ABB RobotStudio station: IndustrialFinal_1.3.rspag

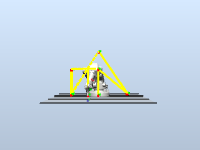
--- station ---
Station IndustrialFinal_1 (saved by RobotStudio 6.5.7558.2005)
Controller IRB_1600_8kg_1.2m
  mechanical unit ROB_1: IRB1600_8_120__02, 6 joints, base frame (0, 0, 0) mm
Layout (positions relative to the parent item):
  - IRB1600_8_120__02 [mechanism, from Robots\IRB1600_8_120_G_02.rslib] at (0, 0, 0) mm; joint values [-0.1857, 1.3903, -0.8163, -2.5988, -0.2555, 2.4812] (rad or m)
  - MyTool [mechanism, from Training Objects\myTool.rslib] at (1147.81, -206.97, 200) mm, rotated rx -180 ry 45 rz -180 deg
Attachment: MyTool is attached to IRB1600_8_120__02 / Link6

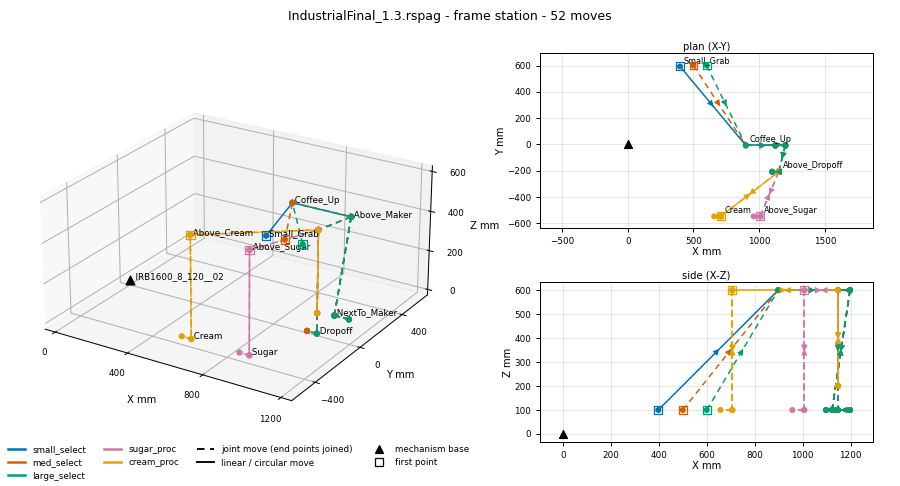
[picture p0: tool path of IndustrialFinal_1.3.rspag in frame station, 52 of 57 moves have a stored position in this frame; points joined in program order, loops and branches not executed]
--- Backups/IRB_1600_8kg_1.2m/RAPID/TASK1/PROGMOD/Module1.mod ---
MODULE Module1
	CONST jointtarget Home_Pos:=[[0,0,0,0,0,0],[9E+09,9E+09,9E+09,9E+09,9E+09,9E+09]];
    !***********************************************************
    !
    ! Module:  Module1
    !
    ! Description:
    !   <Insert description here>
    !
    ! Author: lgstuehrmann
    !
    ! Version: 1.0
    !
    !***********************************************************


    !***********************************************************
    !
    ! Procedure main
    !
    !   This is the entry point of your program
    !
    !***********************************************************
    VAR socketdev server_socket;
    VAR socketdev client_socket;
    VAR num RemotePort;
    VAR string client_ip;
    VAR string receive_string;
    CONST robtarget Small_Grab:=[[397.808,593.034,100],[0.707106781,0,0.707106781,0],[0,0,-1,1],[9E+09,9E+09,9E+09,9E+09,9E+09,9E+09]];
    CONST robtarget Above_Maker:=[[1197.808,-6.966,600],[0.707106781,0,0.707106781,0],[-1,-1,0,1],[9E+09,9E+09,9E+09,9E+09,9E+09,9E+09]];
    CONST robtarget Med_Grab:=[[500,600,100],[0.707106781,0,0.707106781,0],[0,-2,1,0],[9E+09,9E+09,9E+09,9E+09,9E+09,9E+09]];
    CONST robtarget Large_Grab:=[[600,600,100],[0.707106781,0,0.707106781,0],[0,-2,1,0],[9E+09,9E+09,9E+09,9E+09,9E+09,9E+09]];
    CONST robtarget NextTo_Maker:=[[1122.808,-6.966,100],[0.707106781,0,0.707106781,0],[-1,-1,0,1],[9E+09,9E+09,9E+09,9E+09,9E+09,9E+09]];
    CONST robtarget In_Maker:=[[1197.808,-6.966,100],[0.707106781,0,0.707106781,0],[-1,-1,0,1],[9E+09,9E+09,9E+09,9E+09,9E+09,9E+09]];
    CONST robtarget Above_Dropoff:=[[1147.808,-206.966,600],[0.707106781,0,0.707106781,0],[-1,-1,0,1],[9E+09,9E+09,9E+09,9E+09,9E+09,9E+09]];
    CONST robtarget Dropoff:=[[1147.808,-206.966,100],[0.707106781,0,0.707106781,0],[-1,-1,0,1],[9E+09,9E+09,9E+09,9E+09,9E+09,9E+09]];
    CONST robtarget Clearance_Dropoff:=[[1097.808,-206.966,100],[0.707106781,0,0.707106781,0],[-1,-1,0,1],[9E+09,9E+09,9E+09,9E+09,9E+09,9E+09]];
    CONST robtarget Coffee_Up:=[[897.808,-6.966,600],[0.707106781,0,0.707106781,0],[-1,-1,0,1],[9E+09,9E+09,9E+09,9E+09,9E+09,9E+09]];
	CONST robtarget Above_Sugar:=[[1007.019,-546.265,600],[0.707106781,0,0.707106781,0],[-1,1,-2,0],[9E+09,9E+09,9E+09,9E+09,9E+09,9E+09]];
	CONST robtarget Sugar:=[[1007.019,-546.265,100],[0.707106781,0,0.707106781,0],[-1,1,-2,0],[9E+09,9E+09,9E+09,9E+09,9E+09,9E+09]];
	CONST robtarget Pouring_Point:=[[1147.808,-206.966,200],[0.707106781,0,0.707106781,0],[-1,-1,0,1],[9E+09,9E+09,9E+09,9E+09,9E+09,9E+09]];
	CONST robtarget Pour:=[[1147.808,-206.966,200],[0.382683432,0,0.923879533,0],[-1,-2,1,1],[9E+09,9E+09,9E+09,9E+09,9E+09,9E+09]];
	CONST robtarget Clearance_Sugar:=[[957.019,-546.265,100],[0.707106781,0,0.707106781,0],[-1,1,-2,0],[9E+09,9E+09,9E+09,9E+09,9E+09,9E+09]];
	CONST robtarget Above_Cream:=[[707.019,-546.265,600],[0.707106781,0,0.707106781,0],[-1,1,-2,0],[9E+09,9E+09,9E+09,9E+09,9E+09,9E+09]];
	CONST robtarget Cream:=[[707.019,-546.265,100],[0.707106781,0,0.707106781,0],[-1,1,-2,0],[9E+09,9E+09,9E+09,9E+09,9E+09,9E+09]];
	CONST robtarget Clearance_Cream:=[[657.019,-546.265,100],[0.707106781,0,0.707106781,0],[-1,1,-2,0],[9E+09,9E+09,9E+09,9E+09,9E+09,9E+09]];

    !SocketCreate \UDP;


    PROC main()
        !Add your code here

        server_messaging;

        !if small order
        IF receive_string="s" THEN
            !grab from small, fill, & drop off
            small_select;
        ENDIF

        IF receive_string="m" THEN
            !grab from medium, fill, & drop off
            med_select;
        ENDIF

        !if larege order
        IF receive_string="l" THEN
            !grab from large, fill, & drop off
            large_select;
        ENDIF

    ENDPROC


    PROC server_messaging()
        SocketReceive client_socket \str := receive_string;
        SocketSend client_socket \str := "Hello client with ip" + client_ip;
        SocketClose server_socket;
        SocketClose client_socket;
    ERROR
        IF ERRNO=ERR_SOCK_TIMEOUT THEN
        RETRY;

        ELSEIF ERRNO=SOCKET_CLOSED THEN
        server_recover;
        RETRY;
        ELSE
        ! No error recovery handling
        ENDIF
    ENDPROC

    PROC server_recover()

        SocketClose server_socket;
        SocketClose client_socket;
        SocketCreate server_socket;
        SocketBind server_socket, "192.168.0.1", 1025;
        SocketListen server_socket;
        SocketAccept server_socket, client_socket\ClientAddress:=client_ip;
    ERROR
        IF ERRNO=ERR_SOCK_TIMEOUT THEN
        RETRY;
        ELSEIF ERRNO=ERR_SOCK_CLOSED THEN
        RETURN;
        ELSE
        ! No error recovery handling
        ENDIF
    ENDPROC

	PROC small_select()
	    MoveAbsJ Home_Pos,v1000,z100,tool0\WObj:=wobj0;
	    MoveL Small_Grab,v1000,z100,tool0\WObj:=wobj0;
	    MoveL Coffee_Up,v1000,z100,tool0\WObj:=wobj0;
	    MoveL Above_Maker,v1000,z100,tool0\WObj:=wobj0;
	    MoveJ NextTo_Maker,v1000,z100,tool0\WObj:=wobj0;
	    MoveJ In_Maker,v1000,z100,tool0\WObj:=wobj0;
	    MoveJ NextTo_Maker,v1000,z100,tool0\WObj:=wobj0;
	    MoveJ Above_Maker,v1000,z100,tool0\WObj:=wobj0;
	    MoveJ Above_Dropoff,v1000,z100,tool0\WObj:=wobj0;
	    MoveJ Dropoff,v1000,z100,tool0\WObj:=wobj0;
	    MoveJ Clearance_Dropoff,v1000,z100,tool0\WObj:=wobj0;
	ENDPROC

    PROC coffee_select(VAR string s)
        IF s ="1" THEN
            !proc to leave and return to home
        ENDIF

        IF s = "2" THEN
            !proc to sugar
        ENDIF

        IF s = "3" THEN
            !proc to milk
        ENDIF

        IF s = "4" THEN
            !proc to get both
        ENDIF
    ENDPROC
    PROC med_select()
        MoveAbsJ Home_Pos,v1000,z100,tool0\WObj:=wobj0;
        MoveJ Med_Grab,v1000,z100,tool0\WObj:=wobj0;
        MoveJ Coffee_Up,v1000,z100,tool0\WObj:=wobj0;
        MoveJ Above_Maker,v1000,z100,tool0\WObj:=wobj0;
        MoveJ NextTo_Maker,v1000,z100,tool0\WObj:=wobj0;
        MoveJ In_Maker,v1000,z100,tool0\WObj:=wobj0;
        MoveJ NextTo_Maker,v1000,z100,tool0\WObj:=wobj0;
        MoveJ Above_Maker,v1000,z100,tool0\WObj:=wobj0;
        MoveJ Above_Dropoff,v1000,z100,tool0\WObj:=wobj0;
        MoveJ Dropoff,v1000,z100,tool0\WObj:=wobj0;
        MoveJ Clearance_Dropoff,v1000,z100,tool0\WObj:=wobj0;
    ENDPROC
    PROC large_select()
        MoveAbsJ Home_Pos,v1000,z100,tool0\WObj:=wobj0;
        MoveJ Large_Grab,v1000,z100,tool0\WObj:=wobj0;
        MoveJ Coffee_Up,v1000,z100,tool0\WObj:=wobj0;
        MoveJ Above_Maker,v1000,z100,tool0\WObj:=wobj0;
        MoveJ NextTo_Maker,v1000,z100,tool0\WObj:=wobj0;
        MoveJ In_Maker,v1000,z100,tool0\WObj:=wobj0;
        MoveJ NextTo_Maker,v1000,z100,tool0\WObj:=wobj0;
        MoveJ Above_Maker,v1000,z100,tool0\WObj:=wobj0;
        MoveJ Above_Dropoff,v1000,z100,tool0\WObj:=wobj0;
        MoveJ Dropoff,v1000,z100,tool0\WObj:=wobj0;
        MoveJ Clearance_Dropoff,v1000,z100,tool0\WObj:=wobj0;
    ENDPROC
	PROC sugar_proc()
	    MoveJ Above_Sugar,v1000,z100,tool0\WObj:=wobj0;
	    MoveJ Sugar,v1000,z100,tool0\WObj:=wobj0;
	    MoveJ Above_Sugar,v1000,z100,tool0\WObj:=wobj0;
	    MoveJ Above_Dropoff,v1000,z100,tool0\WObj:=wobj0;
	    MoveJ Pouring_Point,v1000,z100,tool0\WObj:=wobj0;
	    MoveJ Pour,v1000,z100,tool0\WObj:=wobj0;
	    MoveJ Pouring_Point,v1000,z100,tool0\WObj:=wobj0;
	    MoveJ Above_Dropoff,v1000,z100,tool0\WObj:=wobj0;
	    MoveJ Above_Sugar,v1000,z100,tool0\WObj:=wobj0;
	    MoveJ Sugar,v1000,z100,tool0\WObj:=wobj0;
	    MoveJ Clearance_Sugar,v1000,z100,tool0\WObj:=wobj0;
	    MoveAbsJ Home_Pos,v1000,z100,tool0\WObj:=wobj0;
	ENDPROC
	PROC cream_proc()
	    MoveJ Above_Cream,v1000,z100,tool0\WObj:=wobj0;
	    MoveJ Cream,v1000,z100,tool0\WObj:=wobj0;
	    MoveJ Above_Cream,v1000,z100,tool0\WObj:=wobj0;
	    MoveJ Above_Dropoff,v1000,z100,tool0\WObj:=wobj0;
	    MoveJ Pouring_Point,v1000,z100,tool0\WObj:=wobj0;
	    MoveJ Pour,v1000,z100,tool0\WObj:=wobj0;
	    MoveJ Pouring_Point,v1000,z100,tool0\WObj:=wobj0;
	    MoveJ Above_Dropoff,v1000,z100,tool0\WObj:=wobj0;
	    MoveJ Above_Cream,v1000,z100,tool0\WObj:=wobj0;
	    MoveJ Cream,v1000,z100,tool0\WObj:=wobj0;
	    MoveJ Clearance_Cream,v1000,z100,tool0\WObj:=wobj0;
	    MoveAbsJ Home_Pos,v1000,z100,tool0\WObj:=wobj0;
	ENDPROC
ENDMODULE

--- Backups/IRB_1600_8kg_1.2m/RAPID/TASK1/SYSMOD/LINKEDM.sys ---
%%%
  VERSION:1
  LANGUAGE:ENGLISH
%%%

MODULE LINKEDM (SYSMODULE)

! FOLLOWER
!     Name of electronically linked follower axis used by operator at teach pendent.
      PERS string l_f_axis_name{5}       :=  ["",  "", "", "", ""];

!     Name of the mechanical unit for follower axis.
      PERS string l_f_mecunt_n{5}  :=  ["", "", "", "", ""];

!     Linked follower axis number in the mechanical unit (first axis in mech. unit is number 1).
      PERS num l_f_axis_no{5}      :=  [0,          0,   0,  0,  0];

! MASTER
!     Name of the mechanical unit for linked master axis.
      PERS string l_m_mecunt_n{5} :=  ["", "", "", "", ""];

!     Linked master axis number in the mechanical unit (first axis in mech. unit is number 1).
!     See axis number table in documentation for different master mechanical units.
      PERS num l_m_axis_no{5}     :=  [0,  0,  0,  0,  0];

! POSITION OFFSET
!     The increase of the allowed offset position between the master and follower
!     positions, used when starting AUTO mode. As soon as the offset is decreased
!     the old configurated parameter is used.
!     Example: 3 => the configurated value of allowed offset is increased 3 times.
      PERS num offset_ratio{5}       :=  [10,  10,   10,  10,  10];

! SPEED RATIO
!     Speed_ratio used in AUTO and JOG modes [ very_slow   slow    normal    fast]
!     Value 1 = max allowed manual speed.
      CONST num speed_ratio {20}      := [0.01, 0.01, 0.01, 0.01, 0.01,
                                          0.05, 0.05, 0.05, 0.05, 0.05,
                                          0.20, 0.20, 0.20, 0.20, 0.20,
                                          1.00, 1.00, 1.00, 1.00, 1.00];

! STEP SIZE
!     Displacement position used in JOG mode for each activation of positive or
!     negative movement.                  [very_short    short   normal   long]
!     Unit degees or meter.
      CONST num displacement {20}     := [0.001, 0.001, 0.001, 0.001, 0.001,
                                          0.005, 0.005, 0.005, 0.005, 0.005,
                                          0.020, 0.020, 0.020, 0.020, 0.020,
                                          0.100, 0.100, 0.100, 0.100, 0.100];


!-------------------------------------------------------------
 PROC Linked_m ()
      Linked_m_exe ;
 ENDPROC
ENDMODULE
